PROGRAM MAIN
VAR
END_VAR

END_PROGRAM

(* stored: Version 1.1.0.1, ProductVersion 3.1.4024.9
   POU MAIN: Id {0e5e8ce8-6958-06d8-3795-06d54b70fbf7}, SpecialFunc None *)
